// TwinCAT 3 PLC project Alarmserver_PLC
// ProgramVersion: 3.1.4023.0
// libraries:
//   Tc2_EtherCAT, * (Beckhoff Automation GmbH)
//   Tc2_Standard, * (Beckhoff Automation GmbH)
//   Tc2_System, * (Beckhoff Automation GmbH)
//   Tc2_Utilities, * (Beckhoff Automation GmbH)
//   Tc3_Database, * (Beckhoff Automation GmbH)
//   Tc3_EventLogger, * (Beckhoff Automation GmbH)
//   Tc3_Module, * (Beckhoff Automation GmbH)
// project tree:
//   DUTs/ Alarms.TcDUT, DUT_AlarmDB.TcDUT
//   / PlcTask.TcTTO
//   POUs/ AlarmServer.TcPOU, EventLogger.TcPOU, FB_Alarm.TcPOU, MAIN.TcPOU
// real-time tasks:
//   TASK PlcTask: cycle T#10ms, priority 20, ADS port 350

CONFIGURATION Alarmserver_PLC
    RESOURCE PLC ON TwinCAT3
        TASK PlcTask(INTERVAL := T#10ms, PRIORITY := 20);
        PROGRAM MAIN WITH PlcTask : MAIN;
    END_RESOURCE
END_CONFIGURATION

// ---- DUTs/Alarms.TcDUT
TYPE Alarms :
STRUCT
	bIsUsed				: BOOL;
	sName				: STRING; 
	bIsActive			: INT;
	bIsAcknowledged		: INT;
	uiID				: UINT;
	sAlarmText			: STRING;
	tActiveStartTime	: STRING;
	tAcknowlegedTime	: STRING;
	tClearedTime		: STRING;
	uiRepeatCount		: DINT;
	
END_STRUCT
END_TYPE

// ---- DUTs/DUT_AlarmDB.TcDUT
TYPE DUT_AlarmDB :
STRUCT
	sname: STRING(255);
	tactivestarttime: STRING(255);
	tacktime: STRING(255);
	tclearedtime: STRING(255);
	uirepeatcount: LINT;
	salarmtext: STRING(255);
	bisactive: LINT;
	bisacknowledged: lINT;
END_STRUCT
END_TYPE

// ---- POUs/MAIN.TcPOU
PROGRAM MAIN
VAR
	Alarms : AlarmServer;	
	Events: Eventlogger;
	Berra: BOOL;
	Baz: BOOL;
	Ack: BOOL;
	clear: BOOL;
	ddd: BOOL;
	
	startTime			: ULINT;
	stopTime			: ULINT;
	diffTime			: ULINT;
	i :INT;	
	AckAll: BOOL;
	READ: BOOL;

	number: INT := 5;
END_VAR

Alarms();
Events();

IF Berra THEN

	startTime:= F_GetActualDcTime64();
	Berra := FALSE;
		
	FOR i:=0 TO number DO 
		Alarms.NewAlarm(sName:=INT_TO_STRING(i), sAlarmText:= 'Ett nytt larm');
	END_FOR
	
	stopTime:= F_GetActualDcTime64();
	diffTime := (stopTime - startTime);
END_IF
IF Baz THEN
	Baz := FALSE;
		
	Alarms.NewAlarm(sName:='Bingo', sAlarmText:= 'Ett nytt larm');
	Alarms.NewAlarm(sName:='Baz', sAlarmText:= 'Ett nytt larm');
	Alarms.NewAlarm(sName:='Tjo', sAlarmText:= 'Ett nytt larm');
	Alarms.NewAlarm(sName:='Tjo', sAlarmText:= 'Bazinga');
END_IF


IF Ack THEN
	startTime:= F_GetActualDcTime64();
	Ack := FALSE;
	Alarms.AckAlarm(iRow:= 900 );
	stopTime:= F_GetActualDcTime64();
	diffTime := (stopTime - startTime);
END_IF

IF AckAll THEN
	startTime:= F_GetActualDcTime64();
	AckAll := FALSE;
	Alarms.AckAllAlarms();
	stopTime:= F_GetActualDcTime64();
	diffTime := (stopTime - startTime);
END_IF

IF clear THEN
	clear := FALSE;
	Alarms.ClearAllAlarms();
END_IF

IF ddd THEN
	ddd := FALSE;
		
	Alarms.NewAlarm(sName:='Braf', sAlarmText:= 'Ett nytt larm');
	Alarms.NewAlarm(sName:='Gizmo', sAlarmText:= 'Ett nytt larm');
END_IF

IF READ THEN
	startTime:= F_GetActualDcTime64();
	READ := FALSE;
	Alarms.ReadFromDB(NrOfRows:= 10);
	stopTime:= F_GetActualDcTime64();
	diffTime := (stopTime - startTime);
END_IF

END_PROGRAM

// ---- POUs/AlarmServer.TcPOU
FUNCTION_BLOCK AlarmServer
VAR CONSTANT
	nrAlarms 			: UINT := 2000;
	//sTable 				: STRING:= '"public"."alarmlog"'; // Important to have extra " " around both DBname and table name. PostgreSQL
	sTable 				: STRING:= 'alarmlog'; // Important to have extra " " around both DBname and table name. SQLite
	//DBID				: UINT	:=1; // PostgreSQL
	DBID				: UINT	:=2; // SQLite
	
	//For read Method
	OrderByColumn		: UINT	:=1; 
	StartIndex			: UINT	:=0;
END_VAR
VAR
	init 				: BOOL:= TRUE;
	ColumnNames     	: ARRAY[0..7] OF STRING(50); // Must be set to 50 char!
	dataReturned 		: ARRAY[0..9] OF Alarms; // Array of the numbers of rows you want to store. 
	fbPLCDBWrite    	: FB_PLCDBWriteEvt(sNetID := '', tTimeout := T#5S);
	tcMessageWrite     	: I_TcMessage;
	fbPLCDBRead    		: FB_PLCDBReadEvt (sNetID := '', tTimeout := T#5S);
	tcMessage    		: I_TcMessage;
END_VAR
VAR PERSISTENT
	AlarmData			: ARRAY [0..nrAlarms] OF Alarms;
	iValueChanged 		: INT;
	irowSelected		: INT;
	bAckAlarm 			: BOOL;
	bAckAllAlarms 		: BOOL;
	bClearAllAlarms 	: BOOL;
END_VAR

// First run, init stuff needed to work
IF init THEN
	// Set columnnames -- Must be the same as in DB
	ColumnNames[0] := 'sname';
	ColumnNames[1] := 'tactivestarttime';
	ColumnNames[2] := 'tacktime';
	ColumnNames[3] := 'tclearedtime';
	ColumnNames[4] := 'uirepeatcount';
	ColumnNames[5] := 'salarmtext';
	ColumnNames[6] := 'bisactive';
	ColumnNames[7] := 'bisacknowledged';

	init:= FALSE;
END_IF



IF(bAckAlarm) THEN
	bAckAlarm:= FALSE;
	AckAlarm(iRow:= irowSelected);
END_IF

IF(bAckAllAlarms) THEN
	bAckAllAlarms:= FALSE;
	AckAllAlarms();
END_IF

IF(bClearAllAlarms) THEN
	bClearAllAlarms:= FALSE;
	ClearAllAlarms();
END_IF

METHOD PUBLIC AckAlarm : BOOL
VAR_INPUT
	iRow: INT;
END_VAR

VAR
	i: UINT;
END_VAR
AlarmData[iRow].bIsAcknowledged:=  BOOL_TO_BYTE(TRUE);
AlarmData[iRow].tAcknowlegedTime :=  DCTIME64_TO_STRING( F_GetActualDcTime64() );

// Update variable for valuechange event
iValueChanged:= iValueChanged +1;
END_METHOD

METHOD PUBLIC AckAllAlarms : BOOL
VAR
	i: UINT;
END_VAR
FOR i:=0 TO nrAlarms BY 1 DO
	
	IF AlarmData[i].bIsUsed THEN
		
		AlarmData[i].bIsAcknowledged:=  BOOL_TO_BYTE(TRUE);
		AlarmData[i].tAcknowlegedTime :=  DCTIME64_TO_STRING( F_GetActualDcTime64() );
		// Update variable for valuechange event
		iValueChanged:= iValueChanged +1;
	END_IF	
END_FOR
END_METHOD

METHOD PUBLIC AddToDb : BOOL
VAR_INPUT
	AlarmData			: Alarms;
END_VAR
VAR


	toDb				: DUT_AlarmDB;
	i:INT;

END_VAR
	
toDb.sname 				:= AlarmData.sName;
toDb.tactivestarttime	:= AlarmData.tActiveStartTime;
toDb.tacktime			:= ALarmData.tAcknowlegedTime;
toDb.tclearedtime		:= AlarmData.tClearedTime;
toDb.uirepeatcount		:= AlarmData.uiRepeatCount;
toDb.salarmtext			:= AlarmData.sAlarmText;
toDb.bisactive			:= AlarmData.bIsActive;
toDb.bisacknowledged	:= AlarmData.bIsAcknowledged;


WHILE NOT fbPLCDBWrite.WriteStruct(
	hDBID:= DBID, 
	sTableName:= sTable, 
	pRecord:= ADR(toDb), 
	cbRecord:= SIZEOF(toDb), 
	pColumnNames:= ADR(ColumnNames) , 
	cbColumnNames:= SIZEOF(ColumnNames)) DO
	i:=1;
END_WHILE




(*


// Write one record to Database 
// Call Functionblock
IF fbPLCDBWrite.WriteStruct(
	hDBID:= DBID, 
	sTableName:= sTable, 
	pRecord:= ADR(toDb), 
	cbRecord:= SIZEOF(toDb), 
	pColumnNames:= ADR(ColumnNames) , 
	cbColumnNames:= SIZEOF(ColumnNames))
THEN
	IF fbPLCDBWrite.bError THEN
		tcMessageWrite := fbPLCDBWrite.ipTcResult;
	END_IF
END_IF
*)
END_METHOD

METHOD PUBLIC ClearAlarm : BOOL
VAR_INPUT
	sName: STRING;
END_VAR

VAR
	i: UINT;
END_VAR


FOR i:=0 TO nrAlarms BY 1 DO
	
	IF AlarmData[i].sName = sName THEN
		AlarmData[i].tClearedTime :=  DCTIME64_TO_STRING( F_GetActualDcTime64());
		AlarmData[i].bIsActive :=  0;
		//AlarmData[i].bIsUsed := FALSE;
		
		// Update variable for valuechange event
		iValueChanged:= iValueChanged +1;
	END_IF
	
END_FOR
END_METHOD

METHOD PUBLIC ClearAllAlarms : BOOL
VAR
	i: UINT;	
END_VAR
FOR i:=0 TO nrAlarms BY 1 DO
	
	IF AlarmData[i].bIsAcknowledged = 1 THEN
		AlarmData[i].tClearedTime :=  DCTIME64_TO_STRING( F_GetActualDcTime64());
		AlarmData[i].bIsActive :=  0;
		//AlarmData[i].bIsUsed := FALSE;
		// Update variable for valuechange event
		iValueChanged:= iValueChanged +1;
	END_IF
	
END_FOR
END_METHOD

METHOD PUBLIC NewAlarm : BOOL
VAR_INPUT
	sName: STRING;
	sAlarmText: STRING;	
END_VAR
VAR
	Alarm: Alarms;
	i: UINT;
	bAlarmExists : BOOL;

	actDC : T_DCTIME64;
    sAct  : STRING;
	
END_VAR
Alarm.sName := sName;
Alarm.sAlarmText := sAlarmText; 
Alarm.bIsActive := 1;
Alarm.bIsUsed := TRUE;
Alarm.tClearedTime := '';

actDC := F_GetActualDcTime64();
sAct  := DCTIME64_TO_STRING( actDC );

Alarm.tActiveStartTime :=  sAct;

FOR i:=0 TO nrAlarms BY 1 DO
	
	IF (AlarmData[i].bIsUsed = TRUE AND AlarmData[i].sName = sName) THEN
		AlarmData[i].uiRepeatCount := AlarmData[i].uiRepeatCount + 1;
		AlarmData[i].tActiveStartTime := Alarm.tActiveStartTime;
		AlarmData[i].tAcknowlegedTime := '';
		AlarmData[i].tClearedTime := '';
		AlarmData[i].bIsAcknowledged := 0;
		bAlarmExists:= TRUE;
		EXIT;
	END_IF
	
END_FOR
 
IF bAlarmExists = FALSE THEN
	
	FOR i:=0 TO SIZEOF(AlarmData) - 1 BY 1 DO
		
		IF (AlarmData[i].bIsUsed = FALSE) THEN
			AlarmData[i] := Alarm;
			EXIT;	
		END_IF
		
	END_FOR
END_IF

// Update variable for valuechange event
iValueChanged:= iValueChanged +1;
END_METHOD

METHOD PUBLIC ReadFromDB : BOOL
VAR_INPUT
	NrOfRows 			: UINT:=10;
END_VAR
VAR
	tcMessageRead	    : I_TcMessage;

	
END_VAR
//	Read rows from the db.  	 
IF fbPLCDBRead.ReadStruct(
	hDBID:= DBID, 
	sTableName:= sTable, 
	pColumnNames:= ADR(ColumnNames), 
	cbColumnNames:= SIZEOF(ColumnNames), 
	sOrderByColumn:= ColumnNames[OrderByColumn], 
	eOrderType:= E_OrderType.ASC, 
	nStartIndex:= StartIndex, 
	nRecordCount:= NrOfRows, 
	pData:= ADR(dataReturned), 
	cbData:= SIZEOF(dataReturned))
THEN

	IF fbPLCDBRead.bError THEN
		tcMessageRead:= fbPLCDBRead.ipTcResult;
	END_IF
END_IF
END_METHOD

END_FUNCTION_BLOCK

// ---- POUs/EventLogger.TcPOU
FUNCTION_BLOCK EventLogger
VAR
    bInit : BOOL := TRUE; 
    bRaise : BOOL := FALSE; 
	bConfirm : BOOL := FALSE; 
	bClear : BOOL := FALSE; 

	newAlarm	: FB_Alarm;
	newWarning	: FB_Alarm;
	event3		: FB_Alarm;
END_VAR


newAlarm(
	Alarm_Event:= TC_EVENTS.WindWings.Encoder_No_Response, 
	bInit:= bInit, 
	bRaise:= bRaise, 
	bConfirm:= bConfirm , 
	bClear:= bClear);


newWarning(
	Alarm_Event:= TC_EVENTS.WindWings.Encoder_Warning, 
	bInit:= bInit, 
	bRaise:= bRaise, 
	bConfirm:= bConfirm , 
	bClear:= bClear);
	
event3(
	Alarm_Event:= TC_EVENTS.WindWings.EventMedNamn3, 
	bInit:= bInit, 
	bRaise:= bRaise, 
	bConfirm:= bConfirm , 
	bClear:= bClear);

	
	bInit := FALSE; 
    bRaise := FALSE; 
	bConfirm := FALSE; 
	bClear := FALSE;

END_FUNCTION_BLOCK

// ---- POUs/FB_Alarm.TcPOU
FUNCTION_BLOCK FB_Alarm
VAR_INPUT
	Alarm_Event: TcEventEntry;
	bInit : BOOL; 
    bRaise : BOOL; 
	bConfirm : BOOL; 
	bClear : BOOL; 
END_VAR
VAR
    fbAlarm : FB_TcAlarm; 
	sALarm : I_TcSourceInfo;
	bConfimed : BOOL;
END_VAR

IF bInit THEN
    bInit := FALSE; 
	bConfimed:= FALSE;
    fbAlarm.CreateEx(Alarm_Event, TRUE, sALarm); 
	fbAlarm.Confirm(0); 
END_IF

IF bRaise THEN 
    bRaise := FALSE; 
    fbAlarm.Raise(0); 
END_IF

IF bConfirm OR fbAlarm.eConfirmationState = 3 THEN
    bConfirm := FALSE; 
	bConfimed:= TRUE;
    fbAlarm.Confirm(0); 
END_IF

IF bClear THEN 
    bClear := FALSE; 
    fbAlarm.Clear(0, TRUE); 
END_IF

END_FUNCTION_BLOCK
